// TIA Portal V15.1 export
// export: Created 2024-06-21T08:40:55.7597518Z, ExportSetting WithDefaults, DisplayName Totally Integrated Automation Portal, DisplayVersion V15.1 Update 5, DisplayName TIA Portal Openness, DisplayVersion V15.1 Update 5, DisplayName SINAMICS Startdrive Advanced, DisplayVersion V15.1, DisplayName G130, G150, S120, S150, SINAMICS MV, S210, DisplayVersion V15.1, DisplayName G110M, G120, G120C, G120D, G120P, DisplayVersion V15.1, DisplayName STEP 7 Professional, DisplayVersion V15.1 Update 5, DisplayName STEP 7 Safety, DisplayVersion V15.1, DisplayName WinCC Professional, DisplayVersion V15.1 Update 5, DisplayName SIMATIC Visualization Architect, DisplayVersion V15.1
FUNCTION "LWeekNumberS7-1500" : Void   // FC2515, SCL
{ S7_Optimized_Access := 'TRUE' }
VERSION : 0.1
// stored: AutoNumber false, IsIECCheckEnabled false, SetENOAutomatically False, UDAEnableTagReadback false
   VAR_OUTPUT
      O_WeekNumber : Int;   // Week number for PLC clock (ISO8601)
   END_VAR
   VAR_TEMP
      iDate : DTL;   // Current date
      SysReturn : Int;   // Return code from RD_SYS_T
      oDate : DInt;   // Current date (as days since 1990-01-01)
      jan1cy : DInt;   // January 1 current year
      wd1jan : Int;   // Weekday of Jan 1
      daycorr : DInt;   // Day correction factor
      yyyy : Int;   // Current year
      wd31dec : Int;   // Weekday of Dec 31
      maxweeks : Int;   // Total number of weeks of current year
      Leap_Year : Bool;   // Leap year
   END_VAR
BEGIN
   (**************************************************************************
   **  This function calculates the calendar week for the current CPU date  **
   **  -------------------------------------------------------------------  **
   **  The calendar week is the return value of the function.               **
   **  The week number is calculated according to DIN 1355 / ISO 8601.      **
   **  "Week no. 1 is the first week, which includes at least four days     **
   **  of the new year. The beginning of a week is always a Monday."        **
   **                                                                       **
   **  The function can be used from year 1991 to 2089.                     **
   **                                                                       **
   **************************************************************************)

   #SysReturn := RD_LOC_T(#iDate); // Get actual date
   #oDate := DATE_TO_DINT(DTL_TO_DATE(#iDate));  // Convert to days since Jan 1 1990

   (* Calculate year including century and days passed since Jan 1 1990 upto Jan 1 current year *)
   #yyyy := DINT_TO_INT(((100 * #oDate) + 50) / 36525) + 1990;
   #jan1cy := ((INT_TO_DINT(#yyyy) * 1461 - 2907389) / 4);

   (* Calculate which day of the week current year started on *)
   #wd1jan := DINT_TO_INT((#jan1cy) MOD 7) + 1;

   (* Correction for weekday of Jan 1 *)
   IF #wd1jan < 5 THEN
       #daycorr := #jan1cy - (#wd1jan + 6);
   ELSE
       #daycorr := #jan1cy - (#wd1jan - 1);
   END_IF;

   (* Week number of current date *)
   #O_WeekNumber := DINT_TO_INT((#oDate - #daycorr) / 7);

   (* Correction when week number equals 0 - Check which week was the last in previous year. *)
   IF #O_WeekNumber = 0 THEN
       IF #wd1jan > 1 THEN
           #wd31dec := #wd1jan - 1;
       ELSE
           #wd31dec := 7;
       END_IF;
       IF #yyyy-1 MOD 400 = 0 THEN
           #Leap_Year := TRUE;
       ELSIF #yyyy-1 MOD 100 = 0 THEN
           #Leap_Year := FALSE;
       ELSIF #yyyy-1 MOD 4 = 0 THEN
           #Leap_Year := TRUE;
       ELSE
           #Leap_Year := FALSE;
       END_IF;
       (* A year usually start and ends on the same weekday, but not on leap years. *)
       IF #Leap_Year AND #wd31dec > 1 THEN
           #wd1jan := #wd31dec - 1;
       ELSE
           #wd1jan := 7;
       END_IF;
       (* If the previous year starts or ends on a Thursday it has 53 weeks. *)
       #O_WeekNumber := 52 + BOOL_TO_INT(#wd31dec = 4 OR #wd1jan = 4);
   ELSE
       IF #yyyy MOD 400 = 0 THEN
           #Leap_Year := TRUE;
       ELSIF #yyyy MOD 100 = 0 THEN
           #Leap_Year := FALSE;
       ELSIF #yyyy MOD 4 = 0 THEN
           #Leap_Year := TRUE;
       ELSE
           #Leap_Year := FALSE;
       END_IF;
       (* A year usually start and ends on the same weekday, but not on leap years. *)
       IF #Leap_Year THEN
           IF #wd1jan < 7 THEN
               #wd31dec := #wd1jan + 1;
           ELSE
               #wd31dec := 1;
           END_IF;
       ELSE
           #wd31dec := #wd1jan;
       END_IF;
       (* Number of weeks current year; if first or last day is thursday then the year has 53 weeks otherwise only 52 *)
       #maxweeks := 52 + BOOL_TO_INT(#wd31dec = 4 OR #wd1jan = 4);
       (* If estimated week number is greater than maximum of current year, it must be the first week of next year *)
       IF #O_WeekNumber > #maxweeks THEN
           #O_WeekNumber := 1;
       END_IF;
   END_IF;
END_FUNCTION
